ABB RAPID module: DEMO_GLOBALPOINT.mod

MODULE DEMO_GLOBALPOINT
const jointtarget P00   := [[0.0, 0.0, 0.0, 0.0, 0.0, 0.0], [0.0, 0.0, 0.0, 0.0, 0.0, 0.0]];

const robtarget Pick01:= [[0.0,0.0,0.0],[0.0,0.0,0.0,0.0],[0,0,0,0],[9E+09,9E+09,9E+09,9E+09,9E+09,9E+09]];
const robtarget Pick02:= [[0.0,0.0,0.0],[0.0,0.0,0.0,0.0],[0,0,0,0],[9E+09,9E+09,9E+09,9E+09,9E+09,9E+09]];
const robtarget Pick03:= [[0.0,0.0,0.0],[0.0,0.0,0.0,0.0],[0,0,0,0],[9E+09,9E+09,9E+09,9E+09,9E+09,9E+09]];
const robtarget Pick04:= [[0.0,0.0,0.0],[0.0,0.0,0.0,0.0],[0,0,0,0],[9E+09,9E+09,9E+09,9E+09,9E+09,9E+09]];
const robtarget Pick05:= [[0.0,0.0,0.0],[0.0,0.0,0.0,0.0],[0,0,0,0],[9E+09,9E+09,9E+09,9E+09,9E+09,9E+09]];
const robtarget Pick06:= [[0.0,0.0,0.0],[0.0,0.0,0.0,0.0],[0,0,0,0],[9E+09,9E+09,9E+09,9E+09,9E+09,9E+09]];
const robtarget Pick07:= [[0.0,0.0,0.0],[0.0,0.0,0.0,0.0],[0,0,0,0],[9E+09,9E+09,9E+09,9E+09,9E+09,9E+09]];
const robtarget Pick08:= [[0.0,0.0,0.0],[0.0,0.0,0.0,0.0],[0,0,0,0],[9E+09,9E+09,9E+09,9E+09,9E+09,9E+09]];
const robtarget Pick09:= [[0.0,0.0,0.0],[0.0,0.0,0.0,0.0],[0,0,0,0],[9E+09,9E+09,9E+09,9E+09,9E+09,9E+09]];
const robtarget Pick10:= [[0.0,0.0,0.0],[0.0,0.0,0.0,0.0],[0,0,0,0],[9E+09,9E+09,9E+09,9E+09,9E+09,9E+09]];

const robtarget Drop01:= [[0.0,0.0,0.0],[0.0,0.0,0.0,0.0],[0,0,0,0],[9E+09,9E+09,9E+09,9E+09,9E+09,9E+09]];
const robtarget Drop02:= [[0.0,0.0,0.0],[0.0,0.0,0.0,0.0],[0,0,0,0],[9E+09,9E+09,9E+09,9E+09,9E+09,9E+09]];
const robtarget Drop03:= [[0.0,0.0,0.0],[0.0,0.0,0.0,0.0],[0,0,0,0],[9E+09,9E+09,9E+09,9E+09,9E+09,9E+09]];
const robtarget Drop04:= [[0.0,0.0,0.0],[0.0,0.0,0.0,0.0],[0,0,0,0],[9E+09,9E+09,9E+09,9E+09,9E+09,9E+09]];
const robtarget Drop05:= [[0.0,0.0,0.0],[0.0,0.0,0.0,0.0],[0,0,0,0],[9E+09,9E+09,9E+09,9E+09,9E+09,9E+09]];
const robtarget Drop06:= [[0.0,0.0,0.0],[0.0,0.0,0.0,0.0],[0,0,0,0],[9E+09,9E+09,9E+09,9E+09,9E+09,9E+09]];
const robtarget Drop07:= [[0.0,0.0,0.0],[0.0,0.0,0.0,0.0],[0,0,0,0],[9E+09,9E+09,9E+09,9E+09,9E+09,9E+09]];
const robtarget Drop08:= [[0.0,0.0,0.0],[0.0,0.0,0.0,0.0],[0,0,0,0],[9E+09,9E+09,9E+09,9E+09,9E+09,9E+09]];
const robtarget Drop09:= [[0.0,0.0,0.0],[0.0,0.0,0.0,0.0],[0,0,0,0],[9E+09,9E+09,9E+09,9E+09,9E+09,9E+09]];
const robtarget Drop10:= [[0.0,0.0,0.0],[0.0,0.0,0.0,0.0],[0,0,0,0],[9E+09,9E+09,9E+09,9E+09,9E+09,9E+09]];

const robtarget MultiProc01:= [[0.0,0.0,0.0],[0.0,0.0,0.0,0.0],[0,0,0,0],[9E+09,9E+09,9E+09,9E+09,9E+09,9E+09]];
const robtarget MultiProc02:= [[0.0,0.0,0.0],[0.0,0.0,0.0,0.0],[0,0,0,0],[9E+09,9E+09,9E+09,9E+09,9E+09,9E+09]];
const robtarget MultiProc03:= [[0.0,0.0,0.0],[0.0,0.0,0.0,0.0],[0,0,0,0],[9E+09,9E+09,9E+09,9E+09,9E+09,9E+09]];
const robtarget MultiProc04:= [[0.0,0.0,0.0],[0.0,0.0,0.0,0.0],[0,0,0,0],[9E+09,9E+09,9E+09,9E+09,9E+09,9E+09]];
const robtarget MultiProc05:= [[0.0,0.0,0.0],[0.0,0.0,0.0,0.0],[0,0,0,0],[9E+09,9E+09,9E+09,9E+09,9E+09,9E+09]];
const robtarget MultiProc06:= [[0.0,0.0,0.0],[0.0,0.0,0.0,0.0],[0,0,0,0],[9E+09,9E+09,9E+09,9E+09,9E+09,9E+09]];
const robtarget MultiProc07:= [[0.0,0.0,0.0],[0.0,0.0,0.0,0.0],[0,0,0,0],[9E+09,9E+09,9E+09,9E+09,9E+09,9E+09]];
const robtarget MultiProc08:= [[0.0,0.0,0.0],[0.0,0.0,0.0,0.0],[0,0,0,0],[9E+09,9E+09,9E+09,9E+09,9E+09,9E+09]];
const robtarget MultiProc09:= [[0.0,0.0,0.0],[0.0,0.0,0.0,0.0],[0,0,0,0],[9E+09,9E+09,9E+09,9E+09,9E+09,9E+09]];
const robtarget MultiProc10:= [[0.0,0.0,0.0],[0.0,0.0,0.0,0.0],[0,0,0,0],[9E+09,9E+09,9E+09,9E+09,9E+09,9E+09]];

const robtarget Proc01:= [[0.0,0.0,0.0],[0.0,0.0,0.0,0.0],[0,0,0,0],[9E+09,9E+09,9E+09,9E+09,9E+09,9E+09]];
const robtarget Proc02:= [[0.0,0.0,0.0],[0.0,0.0,0.0,0.0],[0,0,0,0],[9E+09,9E+09,9E+09,9E+09,9E+09,9E+09]];
const robtarget Proc03:= [[0.0,0.0,0.0],[0.0,0.0,0.0,0.0],[0,0,0,0],[9E+09,9E+09,9E+09,9E+09,9E+09,9E+09]];
const robtarget Proc04:= [[0.0,0.0,0.0],[0.0,0.0,0.0,0.0],[0,0,0,0],[9E+09,9E+09,9E+09,9E+09,9E+09,9E+09]];
const robtarget Proc05:= [[0.0,0.0,0.0],[0.0,0.0,0.0,0.0],[0,0,0,0],[9E+09,9E+09,9E+09,9E+09,9E+09,9E+09]];
const robtarget Proc06:= [[0.0,0.0,0.0],[0.0,0.0,0.0,0.0],[0,0,0,0],[9E+09,9E+09,9E+09,9E+09,9E+09,9E+09]];
const robtarget Proc07:= [[0.0,0.0,0.0],[0.0,0.0,0.0,0.0],[0,0,0,0],[9E+09,9E+09,9E+09,9E+09,9E+09,9E+09]];
const robtarget Proc08:= [[0.0,0.0,0.0],[0.0,0.0,0.0,0.0],[0,0,0,0],[9E+09,9E+09,9E+09,9E+09,9E+09,9E+09]];
const robtarget Proc09:= [[0.0,0.0,0.0],[0.0,0.0,0.0,0.0],[0,0,0,0],[9E+09,9E+09,9E+09,9E+09,9E+09,9E+09]];
const robtarget Proc10:= [[0.0,0.0,0.0],[0.0,0.0,0.0,0.0],[0,0,0,0],[9E+09,9E+09,9E+09,9E+09,9E+09,9E+09]];
ENDMODULE
